// TIA Portal V19 export
DATA_BLOCK "DB_FromHmi"   // DB29
{ S7_Optimized_Access := 'TRUE'; DB_Accessible_From_OPC_UA := 'FALSE' }
// stored: AutoNumber false, DBAccessibleFromOPCUA false, DBAccessibleFromWebserver false, MemoryReserve 100
   VAR
      xLightTest : Bool;   // Light test
      xResetFault : Bool;   // Reset fault and safety
      xStartVacuum : Bool;   // Start vacuum
      xStopVacuum : Bool;   // Stop vacuum
      xReqChangeBigbag : Bool;   // Request change Bigbag
      xValidationBigbagChanged : Bool;   // Validation operator bigbag changed
      xListRecipe : Bool;   // Do the list of all the recipe available in the data base
      xLoadRecipe : Bool;   // Load current recipe from data base
      xSaveRecipe : Bool;   // Save current recipe into the data base
      xNewRecipe : Bool;   // Select next free recipe on the data base
      xDeleteRecipe : Bool;   // Delete the recipe from the data base
      xNextRecipe : Bool;   // Load next recipe in the data base
      xPrevRecipe : Bool;   // Load previus recipe in the data base
      xValideOperation : Bool;   // Validation Operator to remove or Put disk on FerRobotic head
      xValideFault : Bool;   // Validation Operator of Flatness fault
      xProdRecordNext : Bool;
      xProdRecordPrev : Bool;
      xProdRecordDeleteAll : Bool;
      xFlatRecNextLeftRobot : Bool;
      xFlatRecPrevLeftRobot : Bool;
      xFlatRecDelAllLeftRobot : Bool;
      xFlatRecNextRightRobot : Bool;
      xFlatRecPrevRightRobot : Bool;
      xFlatRecDelAllRightRobot : Bool;
   END_VAR
   VAR RETAIN
      xEnableStartLeftRobot : Bool;   // Enable start robot
      xEnableStartRightRobot : Bool;   // Enable start robot
   END_VAR
   VAR
      xDryRun : Bool;   // Robot run in DryRun
      xExportProdData : Bool;
      xExportFlatCtrlRobot1 : Bool;
      xExportFlatCtrlRobot2 : Bool;
      uiCurentRecord : UInt;
      uiFlatCurentRecLeftRobot : UInt;
      uiFlatCurentRecRightRobot : UInt;
      uiDisplayJobNumber : UInt;
   END_VAR
   VAR RETAIN
      usiOperatingMode : USInt;   // Operating mode (1 = Semi-Auto, 2 = Auto)
      uiUserGroup : USInt;   // User grope number logged on HMI
   END_VAR
   VAR
      LeftRobot : Struct   // Command for left robot
         xResetGrafcet : Bool;   // Reset robot communication grafcet
         xStartCycle : Bool;   // Start Cycle
         xStopCycle : Bool;   // Stop Cycle
         xCancelCycle : Bool;   // Cancel cycle
         xStopEndCycle : Bool;   // Stop end of cycle
         xReqChangeDisk : Bool;
         xStartServicePath : Bool;   // Start service path
         xStopServicePath : Bool;   // Stop service path
         xCancelServicePath : Bool;   // Cancel service path
         usiJobNumberDisplay : USInt;   // Job number displayed for robot left
         uiServicePathNumber : UInt;   // Service path number
         xCmdManuLockGimball : Bool;
         xCmdManuLockEccentric1 : Bool;
         xCmdManuLockEccentric2 : Bool;
         xCmdManuLockEccentric3 : Bool;
         xCmdManuEnableRotate : Bool;
         xCmdManuCloseVacValve : Bool;
         xCmdManuOpenVacValve : Bool;
         xCmdManuRemoveConfig : Bool;   // Manual command for activate the Remove config on FerRobotic Head
         xCmdManuPickupConfig : Bool;   // Manual command for activate the Pickup config on FerRobotic Head
         xCmdManuFlatnessConfig : Bool;   // Manual command for activate the Flatness check config on FerRobotic Head
         xMaintStartProg : Bool;
         xMaintStartMain : Bool;
         xForceLubricationX : Bool;
         xForceLubricationZ : Bool;
         ParamManu : "stFerRoboticParam";
      END_STRUCT;
      RightRobot : Struct   // Commande for right robot
         xResetGrafcet : Bool;   // Reset robot communication grafcet
         xStartCycle : Bool;   // Start Cycle
         xStopCycle : Bool;   // Stop Cycle
         xCancelCycle : Bool;   // Cancel cycle
         xStopEndCycle : Bool;   // Stop end of cycle
         xReqChangeDisk : Bool;
         xStartServicePath : Bool;   // Start service path
         xStopServicePath : Bool;   // Stop service path
         xCancelServicePath : Bool;   // Cancel service path
         usiJobNumberDisplay : USInt;   // Job number displayed for robot right
         uiServicePathNumber : UInt;   // Service path number
         xCmdManuLockGimball : Bool;
         xCmdManuLockEccentric1 : Bool;
         xCmdManuLockEccentric2 : Bool;
         xCmdManuLockEccentric3 : Bool;
         xCmdManuEnableRotate : Bool;
         xCmdManuCloseVacValve : Bool;
         xCmdManuOpenVacValve : Bool;
         xCmdManuRemoveConfig : Bool;   // Manual command for activate the Remove config on FerRobotic Head
         xCmdManuPickupConfig : Bool;   // Manual command for activate the Pickup config on FerRobotic Head
         xCmdManuFlatnessConfig : Bool;   // Manual command for activate the Flatness check config on FerRobotic Head
         xMaintStartProg : Bool;
         xMaintStartMain : Bool;
         xForceLubricationX : Bool;
         xForceLubricationZ : Bool;
         ParamManu : "stFerRoboticParam";
      END_STRUCT;
   END_VAR
BEGIN
END_DATA_BLOCK
